	REGION 9 - Report to control block
	    //Xray
	    "FC_EquipmentReport"(iUDT_Status := #sUDT_CommonStatus,
	                         iqUDT_Control := #iqUDT_EquipmentControl);
	    //Outfeed conveyor
	    "FC_EquipmentReport"(iUDT_Status := #sUDT_OutfeedConvCommonStatus,
	                         iqUDT_Control := #iqUDT_EquipmentControl);
	    //Main conveyor
	    "FC_EquipmentReport"(iUDT_Status := #sUDT_MainConvCommonStatus,
	                         iqUDT_Control := #iqUDT_EquipmentControl);
	    // Infeed conveyor
	    "FC_EquipmentReport"(iUDT_Status := #sUDT_InfeedConvCommonStatus,
	                         iqUDT_Control := #iqUDT_EquipmentControl);
	END_REGION
END_FUNCTION_BLOCK

